Staubli VAL3: Control_YesNO.pgx

public program Control_YesNO(string x_sTitle, bool& x_bRes)
begin



  x_bRes=false
  call Control_PanelMd(x_sTitle)
  call Control_BottomS(",,,,,,是,否")

  while true
    switch getKey()

      //F8
      case 278
        x_bRes=false
        cls()
        return
      break
      //F7
      case  277
         x_bRes=true
         cls()
        return
      break
    endSwitch
    delay(0)
  endWhile
end
